// TIA Portal V20 export
VAR_GLOBAL   // PLC tag table "OPC_UA_Method_StatusCodes"
END_VAR
VAR_GLOBAL CONSTANT   // user constants
   OpcUa_Good : DWord := 16#00000000;
   OpcUa_Uncertain : DWord := 16#40000000;
   OpcUa_Bad : DWord := 16#80000000;
   OpcUa_BadUnexpectedError : DWord := 16#80010000;
   OpcUa_BadInternalError : DWord := 16#80020000;
   OpcUa_BadOutOfMemory : DWord := 16#80030000;
   OpcUa_BadResourceUnavailable : DWord := 16#80040000;
   OpcUa_BadCommunicationError : DWord := 16#80050000;
   OpcUa_BadEncodingError : DWord := 16#80060000;
   OpcUa_BadDecodingError : DWord := 16#80070000;
   OpcUa_BadEncodingLimitsExceeded : DWord := 16#80080000;
   OpcUa_BadRequestTooLarge : DWord := 16#80B80000;
   OpcUa_BadResponseTooLarge : DWord := 16#80B90000;
   OpcUa_BadUnknownResponse : DWord := 16#80090000;
   OpcUa_BadTimeout : DWord := 16#800A0000;
   OpcUa_BadServiceUnsupported : DWord := 16#800B0000;
   OpcUa_BadShutdown : DWord := 16#800C0000;
   OpcUa_BadServerNotConnected : DWord := 16#800D0000;
   OpcUa_BadServerHalted : DWord := 16#800E0000;
   OpcUa_BadNothingToDo : DWord := 16#800F0000;
   OpcUa_BadTooManyOperations : DWord := 16#80100000;
   OpcUa_BadTooManyMonitoredItems : DWord := 16#80DB0000;
   OpcUa_BadDataTypeIdUnknown : DWord := 16#80110000;
   OpcUa_BadCertificateInvalid : DWord := 16#80120000;
   OpcUa_BadSecurityChecksFailed : DWord := 16#80130000;
   OpcUa_BadCertificateTimeInvalid : DWord := 16#80140000;
   OpcUa_BadCertificateIssuerTimeInvalid : DWord := 16#80150000;
   OpcUa_BadCertificateHostNameInvalid : DWord := 16#80160000;
   OpcUa_BadCertificateUriInvalid : DWord := 16#80170000;
   OpcUa_BadCertificateUseNotAllowed : DWord := 16#80180000;
   OpcUa_BadCertificateIssuerUseNotAllowed : DWord := 16#80190000;
   OpcUa_BadCertificateUntrusted : DWord := 16#801A0000;
   OpcUa_BadCertificateRevocationUnknown : DWord := 16#801B0000;
   OpcUa_BadCertificateIssuerRevocationUnknown : DWord := 16#801C0000;
   OpcUa_BadCertificateRevoked : DWord := 16#801D0000;
   OpcUa_BadCertificateIssuerRevoked : DWord := 16#801E0000;
   OpcUa_BadCertificateChainIncomplete : DWord := 16#810D0000;
   OpcUa_BadUserAccessDenied : DWord := 16#801F0000;
   OpcUa_BadIdentityTokenInvalid : DWord := 16#80200000;
   OpcUa_BadIdentityTokenRejected : DWord := 16#80210000;
   OpcUa_BadSecureChannelIdInvalid : DWord := 16#80220000;
   OpcUa_BadInvalidTimestamp : DWord := 16#80230000;
   OpcUa_BadNonceInvalid : DWord := 16#80240000;
   OpcUa_BadSessionIdInvalid : DWord := 16#80250000;
   OpcUa_BadSessionClosed : DWord := 16#80260000;
   OpcUa_BadSessionNotActivated : DWord := 16#80270000;
   OpcUa_BadSubscriptionIdInvalid : DWord := 16#80280000;
   OpcUa_BadRequestHeaderInvalid : DWord := 16#802A0000;
   OpcUa_BadTimestampsToReturnInvalid : DWord := 16#802B0000;
   OpcUa_BadRequestCancelledByClient : DWord := 16#802C0000;
   OpcUa_BadTooManyArguments : DWord := 16#80E50000;
   OpcUa_BadLicenseExpired : DWord := 16#810E0000;
   OpcUa_BadLicenseLimitsExceeded : DWord := 16#810F0000;
   OpcUa_BadLicenseNotAvailable : DWord := 16#81100000;
   OpcUa_GoodSubscriptionTransferred : DWord := 16#002D0000;
   OpcUa_GoodCompletesAsynchronously : DWord := 16#002E0000;
   OpcUa_GoodOverload : DWord := 16#002F0000;
   OpcUa_GoodClamped : DWord := 16#00300000;
   OpcUa_BadNoCommunication : DWord := 16#80310000;
   OpcUa_BadWaitingForInitialData : DWord := 16#80320000;
   OpcUa_BadNodeIdInvalid : DWord := 16#80330000;
   OpcUa_BadNodeIdUnknown : DWord := 16#80340000;
   OpcUa_BadAttributeIdInvalid : DWord := 16#80350000;
   OpcUa_BadIndexRangeInvalid : DWord := 16#80360000;
   OpcUa_BadIndexRangeNoData : DWord := 16#80370000;
   OpcUa_BadDataEncodingInvalid : DWord := 16#80380000;
   OpcUa_BadDataEncodingUnsupported : DWord := 16#80390000;
   OpcUa_BadNotReadable : DWord := 16#803A0000;
   OpcUa_BadNotWritable : DWord := 16#803B0000;
   OpcUa_BadOutOfRange : DWord := 16#803C0000;
   OpcUa_BadNotSupported : DWord := 16#803D0000;
   OpcUa_BadNotFound : DWord := 16#803E0000;
   OpcUa_BadObjectDeleted : DWord := 16#803F0000;
   OpcUa_BadNotImplemented : DWord := 16#80400000;
   OpcUa_BadMonitoringModeInvalid : DWord := 16#80410000;
   OpcUa_BadMonitoredItemIdInvalid : DWord := 16#80420000;
   OpcUa_BadMonitoredItemFilterInvalid : DWord := 16#80430000;
   OpcUa_BadMonitoredItemFilterUnsupported : DWord := 16#80440000;
   OpcUa_BadFilterNotAllowed : DWord := 16#80450000;
   OpcUa_BadStructureMissing : DWord := 16#80460000;
   OpcUa_BadEventFilterInvalid : DWord := 16#80470000;
   OpcUa_BadContentFilterInvalid : DWord := 16#80480000;
   OpcUa_BadFilterOperatorInvalid : DWord := 16#80C10000;
   OpcUa_BadFilterOperatorUnsupported : DWord := 16#80C20000;
   OpcUa_BadFilterOperandCountMismatch : DWord := 16#80C30000;
   OpcUa_BadFilterOperandInvalid : DWord := 16#80490000;
   OpcUa_BadFilterElementInvalid : DWord := 16#80C40000;
   OpcUa_BadFilterLiteralInvalid : DWord := 16#80C50000;
   OpcUa_BadContinuationPointInvalid : DWord := 16#804A0000;
   OpcUa_BadNoContinuationPoints : DWord := 16#804B0000;
   OpcUa_BadReferenceTypeIdInvalid : DWord := 16#804C0000;
   OpcUa_BadBrowseDirectionInvalid : DWord := 16#804D0000;
   OpcUa_BadNodeNotInView : DWord := 16#804E0000;
   OpcUa_BadNumericOverflow : DWord := 16#81120000;
   OpcUa_BadServerUriInvalid : DWord := 16#804F0000;
   OpcUa_BadServerNameMissing : DWord := 16#80500000;
   OpcUa_BadDiscoveryUrlMissing : DWord := 16#80510000;
   OpcUa_BadSempahoreFileMissing : DWord := 16#80520000;
   OpcUa_BadRequestTypeInvalid : DWord := 16#80530000;
   OpcUa_BadSecurityModeRejected : DWord := 16#80540000;
   OpcUa_BadSecurityPolicyRejected : DWord := 16#80550000;
   OpcUa_BadTooManySessions : DWord := 16#80560000;
   OpcUa_BadUserSignatureInvalid : DWord := 16#80570000;
   OpcUa_BadApplicationSignatureInvalid : DWord := 16#80580000;
   OpcUa_BadNoValidCertificates : DWord := 16#80590000;
   OpcUa_BadIdentityChangeNotSupported : DWord := 16#80C60000;
   OpcUa_BadRequestCancelledByRequest : DWord := 16#805A0000;
   OpcUa_BadParentNodeIdInvalid : DWord := 16#805B0000;
   OpcUa_BadReferenceNotAllowed : DWord := 16#805C0000;
   OpcUa_BadNodeIdRejected : DWord := 16#805D0000;
   OpcUa_BadNodeIdExists : DWord := 16#805E0000;
   OpcUa_BadNodeClassInvalid : DWord := 16#805F0000;
   OpcUa_BadBrowseNameInvalid : DWord := 16#80600000;
   OpcUa_BadBrowseNameDuplicated : DWord := 16#80610000;
   OpcUa_BadNodeAttributesInvalid : DWord := 16#80620000;
   OpcUa_BadTypeDefinitionInvalid : DWord := 16#80630000;
   OpcUa_BadSourceNodeIdInvalid : DWord := 16#80640000;
   OpcUa_BadTargetNodeIdInvalid : DWord := 16#80650000;
   OpcUa_BadDuplicateReferenceNotAllowed : DWord := 16#80660000;
   OpcUa_BadInvalidSelfReference : DWord := 16#80670000;
   OpcUa_BadReferenceLocalOnly : DWord := 16#80680000;
   OpcUa_BadNoDeleteRights : DWord := 16#80690000;
   OpcUa_UncertainReferenceNotDeleted : DWord := 16#40BC0000;
   OpcUa_BadServerIndexInvalid : DWord := 16#806A0000;
   OpcUa_BadViewIdUnknown : DWord := 16#806B0000;
   OpcUa_BadViewTimestampInvalid : DWord := 16#80C90000;
   OpcUa_BadViewParameterMismatch : DWord := 16#80CA0000;
   OpcUa_BadViewVersionInvalid : DWord := 16#80CB0000;
   OpcUa_UncertainNotAllNodesAvailable : DWord := 16#40C00000;
   OpcUa_GoodResultsMayBeIncomplete : DWord := 16#00BA0000;
   OpcUa_BadNotTypeDefinition : DWord := 16#80C80000;
   OpcUa_UncertainReferenceOutOfServer : DWord := 16#406C0000;
   OpcUa_BadTooManyMatches : DWord := 16#806D0000;
   OpcUa_BadQueryTooComplex : DWord := 16#806E0000;
   OpcUa_BadNoMatch : DWord := 16#806F0000;
   OpcUa_BadMaxAgeInvalid : DWord := 16#80700000;
   OpcUa_BadSecurityModeInsufficient : DWord := 16#80E60000;
   OpcUa_BadHistoryOperationInvalid : DWord := 16#80710000;
   OpcUa_BadHistoryOperationUnsupported : DWord := 16#80720000;
   OpcUa_BadInvalidTimestampArgument : DWord := 16#80BD0000;
   OpcUa_BadWriteNotSupported : DWord := 16#80730000;
   OpcUa_BadTypeMismatch : DWord := 16#80740000;
   OpcUa_BadMethodInvalid : DWord := 16#80750000;
   OpcUa_BadArgumentsMissing : DWord := 16#80760000;
   OpcUa_BadNotExecutable : DWord := 16#81110000;
   OpcUa_BadTooManySubscriptions : DWord := 16#80770000;
   OpcUa_BadTooManyPublishRequests : DWord := 16#80780000;
   OpcUa_BadNoSubscription : DWord := 16#80790000;
   OpcUa_BadSequenceNumberUnknown : DWord := 16#807A0000;
   OpcUa_BadMessageNotAvailable : DWord := 16#807B0000;
   OpcUa_BadInsufficientClientProfile : DWord := 16#807C0000;
   OpcUa_BadStateNotActive : DWord := 16#80BF0000;
   OpcUa_BadTcpServerTooBusy : DWord := 16#807D0000;
   OpcUa_BadTcpMessageTypeInvalid : DWord := 16#807E0000;
   OpcUa_BadTcpSecureChannelUnknown : DWord := 16#807F0000;
   OpcUa_BadTcpMessageTooLarge : DWord := 16#80800000;
   OpcUa_BadTcpNotEnoughResources : DWord := 16#80810000;
   OpcUa_BadTcpInternalError : DWord := 16#80820000;
   OpcUa_BadTcpEndpointUrlInvalid : DWord := 16#80830000;
   OpcUa_BadRequestInterrupted : DWord := 16#80840000;
   OpcUa_BadRequestTimeout : DWord := 16#80850000;
   OpcUa_BadSecureChannelClosed : DWord := 16#80860000;
   OpcUa_BadSecureChannelTokenUnknown : DWord := 16#80870000;
   OpcUa_BadSequenceNumberInvalid : DWord := 16#80880000;
   OpcUa_BadProtocolVersionUnsupported : DWord := 16#80BE0000;
   OpcUa_BadConfigurationError : DWord := 16#80890000;
   OpcUa_BadNotConnected : DWord := 16#808A0000;
   OpcUa_BadDeviceFailure : DWord := 16#808B0000;
   OpcUa_BadSensorFailure : DWord := 16#808C0000;
   OpcUa_BadOutOfService : DWord := 16#808D0000;
   OpcUa_BadDeadbandFilterInvalid : DWord := 16#808E0000;
   OpcUa_UncertainNoCommunicationLastUsableValue : DWord := 16#408F0000;
   OpcUa_UncertainLastUsableValue : DWord := 16#40900000;
   OpcUa_UncertainSubstituteValue : DWord := 16#40910000;
   OpcUa_UncertainInitialValue : DWord := 16#40920000;
   OpcUa_UncertainSensorNotAccurate : DWord := 16#40930000;
   OpcUa_UncertainEngineeringUnitsExceeded : DWord := 16#40940000;
   OpcUa_UncertainSubNormal : DWord := 16#40950000;
   OpcUa_GoodLocalOverride : DWord := 16#00960000;
   OpcUa_BadRefreshInProgress : DWord := 16#80970000;
   OpcUa_BadConditionAlreadyDisabled : DWord := 16#80980000;
   OpcUa_BadConditionAlreadyEnabled : DWord := 16#80CC0000;
   OpcUa_BadConditionDisabled : DWord := 16#80990000;
   OpcUa_BadEventIdUnknown : DWord := 16#809A0000;
   OpcUa_BadEventNotAcknowledgeable : DWord := 16#80BB0000;
   OpcUa_BadDialogNotActive : DWord := 16#80CD0000;
   OpcUa_BadDialogResponseInvalid : DWord := 16#80CE0000;
   OpcUa_BadConditionBranchAlreadyAcked : DWord := 16#80CF0000;
   OpcUa_BadConditionBranchAlreadyConfirmed : DWord := 16#80D00000;
   OpcUa_BadConditionAlreadyShelved : DWord := 16#80D10000;
   OpcUa_BadConditionNotShelved : DWord := 16#80D20000;
   OpcUa_BadShelvingTimeOutOfRange : DWord := 16#80D30000;
   OpcUa_BadNoData : DWord := 16#809B0000;
   OpcUa_BadBoundNotFound : DWord := 16#80D70000;
   OpcUa_BadBoundNotSupported : DWord := 16#80D80000;
   OpcUa_BadDataLost : DWord := 16#809D0000;
   OpcUa_BadDataUnavailable : DWord := 16#809E0000;
   OpcUa_BadEntryExists : DWord := 16#809F0000;
   OpcUa_BadNoEntryExists : DWord := 16#80A00000;
   OpcUa_BadTimestampNotSupported : DWord := 16#80A10000;
   OpcUa_GoodEntryInserted : DWord := 16#00A20000;
   OpcUa_GoodEntryReplaced : DWord := 16#00A30000;
   OpcUa_UncertainDataSubNormal : DWord := 16#40A40000;
   OpcUa_GoodNoData : DWord := 16#00A50000;
   OpcUa_GoodMoreData : DWord := 16#00A60000;
   OpcUa_BadAggregateListMismatch : DWord := 16#80D40000;
   OpcUa_BadAggregateNotSupported : DWord := 16#80D50000;
   OpcUa_BadAggregateInvalidInputs : DWord := 16#80D60000;
   OpcUa_BadAggregateConfigurationRejected : DWord := 16#80DA0000;
   OpcUa_GoodDataIgnored : DWord := 16#00D90000;
   OpcUa_BadRequestNotAllowed : DWord := 16#80E40000;
   OpcUa_BadRequestNotComplete : DWord := 16#81130000;
   OpcUa_GoodEdited : DWord := 16#00DC0000;
   OpcUa_GoodPostActionFailed : DWord := 16#00DD0000;
   OpcUa_UncertainDominantValueChanged : DWord := 16#40DE0000;
   OpcUa_GoodDependentValueChanged : DWord := 16#00E00000;
   OpcUa_BadDominantValueChanged : DWord := 16#80E10000;
   OpcUa_UncertainDependentValueChanged : DWord := 16#40E20000;
   OpcUa_BadDependentValueChanged : DWord := 16#80E30000;
   OpcUa_GoodCommunicationEvent : DWord := 16#00A70000;
   OpcUa_GoodShutdownEvent : DWord := 16#00A80000;
   OpcUa_GoodCallAgain : DWord := 16#00A90000;
   OpcUa_GoodNonCriticalTimeout : DWord := 16#00AA0000;
   OpcUa_BadInvalidArgument : DWord := 16#80AB0000;
   OpcUa_BadConnectionRejected : DWord := 16#80AC0000;
   OpcUa_BadDisconnect : DWord := 16#80AD0000;
   OpcUa_BadConnectionClosed : DWord := 16#80AE0000;
   OpcUa_BadInvalidState : DWord := 16#80AF0000;
   OpcUa_BadEndOfStream : DWord := 16#80B00000;
   OpcUa_BadNoDataAvailable : DWord := 16#80B10000;
   OpcUa_BadWaitingForResponse : DWord := 16#80B20000;
   OpcUa_BadOperationAbandoned : DWord := 16#80B30000;
   OpcUa_BadExpectedStreamToBlock : DWord := 16#80B40000;
   OpcUa_BadWouldBlock : DWord := 16#80B50000;
   OpcUa_BadSyntaxError : DWord := 16#80B60000;
   OpcUa_BadMaxConnectionsReached : DWord := 16#80B70000;
END_VAR
